// TIA Portal V20 export
TYPE "UDT_HMI"
   STRUCT
      NumMesa_Pedida : UInt;   // Numero de Mesa que Pedida por la Pantalla
      PosUT_Tratada : UInt;   // Posición de la UT en la mesa que se Visualiza
      NumMesa_Tratada : UInt;   // Numero de Mesa que se visuliza
      Ordenes_HMI_Mesa { S7_SetPoint := 'True'} : "UDT_ProtocoloRecDispositivo";   // Ordenes para el Dispositivo Mesa
      BitsAviso_HMI_Mesa { S7_SetPoint := 'True'} : "Avisos_HMI_Mesa";   // Bits de Aviso hacia la Mesa
      NumMesa_CambiarUT : UInt;   // Numero de Mesa donde hay que Cambiar la UT
      BitsAviso_Mesa_HMI { S7_SetPoint := 'True'} : "Avisos_Mesa_HMI";   // Bits de Aviso hacia la Pantalla
      TipoMesa { S7_SetPoint := 'True'} : "TipoMesaPantalla";   // Tipo de Mesa para configurar la pantalla
      TMP_Inactividad : UInt;   // Tiempo sin tocar pantalla con mesa bloqueada
      TMP_SinCambiarUT : UDInt;
      Zona_Mesa { S7_SetPoint := 'True'} : "EstadoZona";   // Estado de la Zona de Mesa
      Zona_Maquina { S7_SetPoint := 'True'} : "EstadoZona";   // Estado de la Zona de Maquina
      Estado_Mesa { S7_SetPoint := 'True'} : "EstadosMesa";   // Estado del VI en la Mesa
      Estado_Maquina { S7_SetPoint := 'True'} : "EstadoMaquina";   // Estado del VI en la Maquina
      MoviManual_Mesa { S7_SetPoint := 'True'} : "MoviManualMesa";   // Movimientos Manuales de la Mesa
      MoviManual_Maquinas { S7_SetPoint := 'True'} : "MoviManualMaquina";   // Movimientos Manuales de la Maquina
      Datos_UTs : Struct
         UT_Control { S7_SetPoint := 'True'} : "UDT_UTs_Control";
         UT_Ruta { S7_SetPoint := 'True'} : "UDT_UTs_Ruta";
         UT_TextoPantalla { S7_SetPoint := 'True'} : "UDT_UTs_TextoPantalla";
         UT_Etiqueta { S7_SetPoint := 'True'} : "UDT_UTs_Etiqueta";
         UT_Datos { S7_SetPoint := 'True'} : "UDT_UTs_Datos";
      END_STRUCT;
      Interlock : "UDT_Interlock_generico";
      Interlock_manual { S7_SetPoint := 'True'} : "UDT_Interlock_manual";
   END_STRUCT;
END_TYPE
